{attribute 'GeneratedUsingTerminal: EL6201-0000-0017'}
{attribute addProperty BoxType "EL6201-0000-0017"}
{attribute addProperty Id "Slave_3A_DI0BOOL1Slave_3A_DI1BOOL1Slave_3A_DI2BOOL1Slave_3A_DI3BOOL1Slave_3B_DI0BOOL1Slave_3B_DI1BOOL1Slave_3B_DI2BOOL1Slave_3B_DI3BOOL1"}
{attribute addProperty CRC "2575648125"}
{attribute addProperty Size "8"}
TYPE Slave_3_Inputs_9985457D :
STRUCT
	{attribute addProperty Name "Slave_3A_DI0"}
	Slave_3A_DI0 : BOOL;
	{attribute addProperty Name "Slave_3A_DI1"}
	Slave_3A_DI1 : BOOL;
	{attribute addProperty Name "Slave_3A_DI2"}
	Slave_3A_DI2 : BOOL;
	{attribute addProperty Name "Slave_3A_DI3"}
	Slave_3A_DI3 : BOOL;
	{attribute addProperty Name "Slave_3B_DI0"}
	Slave_3B_DI0 : BOOL;
	{attribute addProperty Name "Slave_3B_DI1"}
	Slave_3B_DI1 : BOOL;
	{attribute addProperty Name "Slave_3B_DI2"}
	Slave_3B_DI2 : BOOL;
	{attribute addProperty Name "Slave_3B_DI3"}
	Slave_3B_DI3 : BOOL;
END_STRUCT
END_TYPE

(* stored: Version 1.2.0.0, ProductVersion 3.1.4024.9
   DUT Slave_3_Inputs_9985457D: Id {f293cdfb-0769-4f8c-bdde-4136b1b832bc} *)
